{attribute 'qualified_only'}
{attribute 'strict'}
{attribute 'to_string'}
TYPE eTcaWorkpiecePlaceShape :
(
	undefined := 0,
	roll,
	ring,
	plate,
	other,
	
	MAXSIZE
);
END_TYPE

(* stored: Version 1.1.0.1
   DUT eTcaWorkpiecePlaceShape: Id {0f1e2cd2-98c8-4828-9139-8246e72a9f1e} *)
